(* CODESYS project Patterns of Ladderlogic programming.project

Project tree, tasks and I/O mapping:
  Device : CODESYS Control for Raspberry Pi SL, 3S - Smart Software Solutions GmbH, version 3.5.12.30
    application Application
      libraries: Standard, * (System); Util, * (System)
      task MainTask (cyclic, interval 50 ms, priority 1) calls PLC_PRG
      program PLC_PRG [LD]
      Ladder Patterns/
        Debounce/
          function block FbDebounce [LD]
        Five Rung/
          function block FbFiveRung [LD]
        Mode/
          function block FbMode [LD]
        Flasher/
          function block FbFlasher [LD]
        Mission/
          function block FbMission [LD]
        Set Reset/
          function block FbSetReset [LD]
        Reset Set/
          function block FbResetSet [LD]
        Sealed In Coil/
          function block FbSealedinCoil [LD]
        Start Stop Circuit/
          function block FbStartStopCircuit [LD]
        Input Map/
          function block FbInputMap [LD]
        State Coil Fault Coil/
          function block FbStateCoilFaultCoil [LD]
        Step/
          function block fbStep [LD]
    SoftMotion General Axis Pool
    I²C
    SPI
    GPIOs_A_B : GPIOs A/B, 3S - Smart Software Solutions GmbH, version 3.5.11.0
        unmapped channels: digital inputs (GPIO0..GPIO31), digital outputs (GPIO0..GPIO31)
    Onewire
    Camera device
      <Empty>
*)

// Device/Application/PLC_PRG
PROGRAM PLC_PRG
VAR
	SealedinCoil : FbSealedinCoil;
	xTrigger : BOOL;
	xSealedInCoil :  BOOL;
	
	
	StateCoilFaultCoil : FbStateCoilFaultCoil;
	xBreakCondition : BOOL;
	xMemoryCoil : BOOL;
	
	
	StartStopCircuit :  FbStartStopCircuit;
	xStart : BOOL;
	xStop: BOOL;
	
	
	SetReset : FbSetReset; (* use SR instead *)
	xRun : BOOL;
	xSet : BOOL;
	
	
	ResetSet : FbResetSet; (* use RS instead *)
	xReset: BOOL;
	xQs: BOOL;
	xQr: BOOL;
	
	Flasher : FbFlasher; (* use BLINK instead *)
	xFlashingLight: BOOL;
	
	
	Debounce : FbDebounce;
	xInput: BOOL;
	xInputDebounced : BOOL;
	
	
	ExtendCylinder : fbStep;
	xExtendCylinderCmd : BOOL;
	TONExtendCylinderDone : TON;
	xExtendCylinderDone: BOOL;
	tETExtend: TIME;
	RetractCylinder : fbStep;
	xRetractCylinderCmd: BOOL;
	TONRetractCylinderDone: TON;
	tETRetract: TIME;
	
	Mission : FbMission;
	xMission1Start : BOOL;
	xMission2Start : BOOL;
	xMission1Done : BOOL;
	xMission2Done : BOOL;
	xNoMission : BOOL;
	xMission1Busy : BOOL;
	xMission2Busy : BOOL;
	
	FiveRung : fbFiveRung;
	xFromSeqLogic: BOOL;
	xEStopOK: BOOL;
	xAutoMode: BOOL;
	xManMode : BOOL;
	xPushButton: BOOL;
	xSensor : BOOL;
	xResetFault: BOOL;
	xTriggerf: BOOL;
	xSafe: BOOL;
	xCommand: BOOL;
	xInPosition: BOOL;
	xTimeoutFault: BOOL;
	
	Mode : FbMode;
	xAutoModePB : BOOL;
	xManModePB : BOOL;
	xAutoSelected :BOOL;
	xManualSelected :BOOL;
	
END_VAR

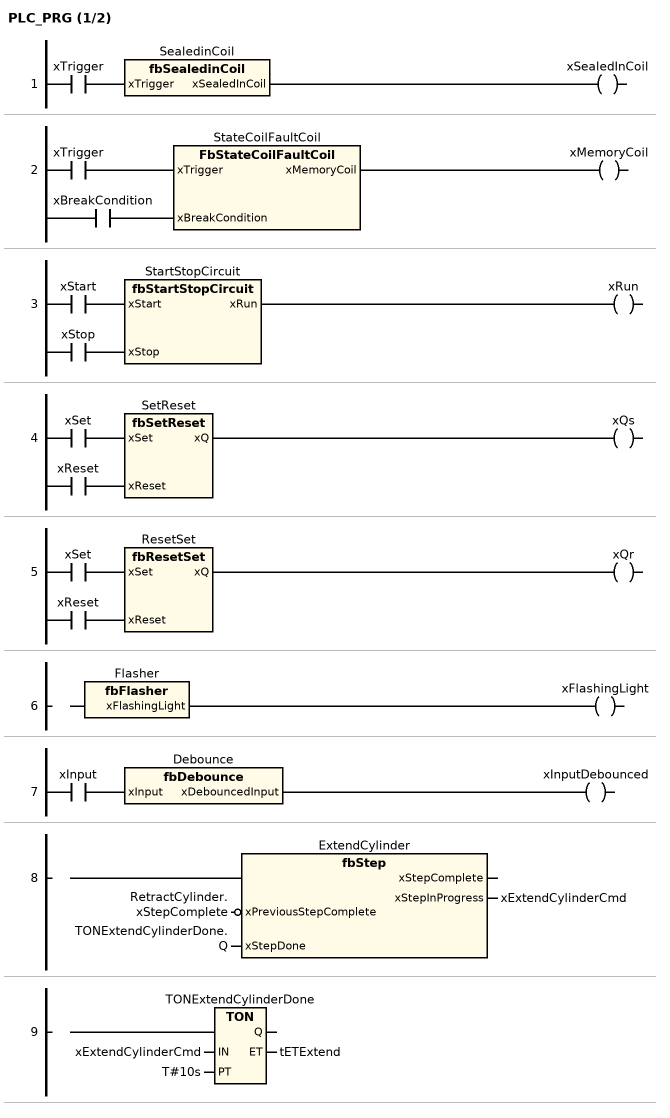
// NETWORK 1
SealedinCoil(xTrigger := xTrigger); // fbSealedinCoil
xSealedInCoil := SealedinCoil.xSealedInCoil;

// NETWORK 2
StateCoilFaultCoil(xTrigger := xTrigger, xBreakCondition := xBreakCondition); // FbStateCoilFaultCoil
xMemoryCoil := StateCoilFaultCoil.xMemoryCoil;

// NETWORK 3
StartStopCircuit(xStart := xStart, xStop := xStop); // fbStartStopCircuit
xRun := StartStopCircuit.xRun;

// NETWORK 4
SetReset(xSet := xSet, xReset := xReset); // fbSetReset
xQs := SetReset.xQ;

// NETWORK 5
ResetSet(xSet := xSet, xReset := xReset); // fbResetSet
xQr := ResetSet.xQ;

// NETWORK 6
Flasher(); // fbFlasher
xFlashingLight := Flasher.xFlashingLight;

// NETWORK 7
Debounce(xInput := xInput); // fbDebounce
xInputDebounced := Debounce.xDebouncedInput;

// NETWORK 8
ExtendCylinder(
    xPreviousStepComplete := NOT RetractCylinder.xStepComplete,
    xStepDone := TONExtendCylinderDone.Q,
    xStepInProgress => xExtendCylinderCmd); // fbStep

// NETWORK 9
TONExtendCylinderDone(IN := xExtendCylinderCmd, PT := T#10s, ET => tETExtend); // TON

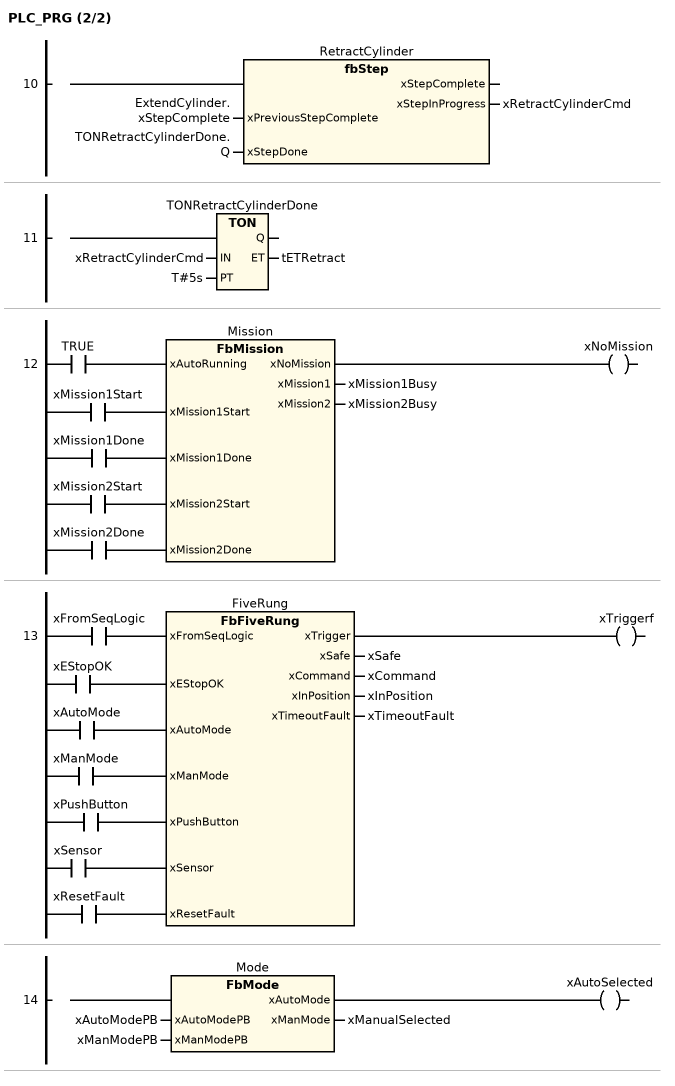
// NETWORK 10
RetractCylinder(
    xPreviousStepComplete := ExtendCylinder.xStepComplete,
    xStepDone := TONRetractCylinderDone.Q,
    xStepInProgress => xRetractCylinderCmd); // fbStep

// NETWORK 11
TONRetractCylinderDone(IN := xRetractCylinderCmd, PT := T#5s, ET => tETRetract); // TON

// NETWORK 12
Mission(
    xAutoRunning := TRUE,
    xMission1Start := xMission1Start,
    xMission1Done := xMission1Done,
    xMission2Start := xMission2Start,
    xMission2Done := xMission2Done,
    xMission1 => xMission1Busy,
    xMission2 => xMission2Busy); // FbMission
xNoMission := Mission.xNoMission;

// NETWORK 13
FiveRung(
    xFromSeqLogic := xFromSeqLogic,
    xEStopOK := xEStopOK,
    xAutoMode := xAutoMode,
    xManMode := xManMode,
    xPushButton := xPushButton,
    xSensor := xSensor,
    xResetFault := xResetFault,
    xSafe => xSafe,
    xCommand => xCommand,
    xInPosition => xInPosition,
    xTimeoutFault => xTimeoutFault); // FbFiveRung
xTriggerf := FiveRung.xTrigger;

// NETWORK 14
Mode(xAutoModePB := xAutoModePB, xManModePB := xManModePB, xManMode => xManualSelected); // FbMode
xAutoSelected := Mode.xAutoMode;

END_PROGRAM

// Device/Application/Ladder Patterns/Sealed In Coil/FbSealedinCoil
FUNCTION_BLOCK FbSealedinCoil
VAR_INPUT	
	xTrigger : BOOL;
END_VAR	
VAR_OUTPUT
	xSealedInCoil : BOOL;	
END_VAR

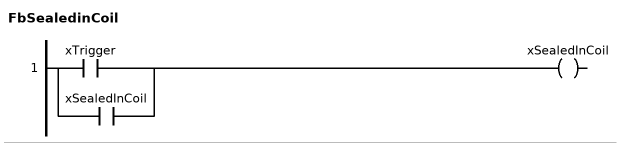
// NETWORK 1
xSealedInCoil := xTrigger OR xSealedInCoil;

END_FUNCTION_BLOCK

// Device/Application/Ladder Patterns/State Coil Fault Coil/FbStateCoilFaultCoil
FUNCTION_BLOCK FbStateCoilFaultCoil
VAR_INPUT
	xTrigger : BOOL;
	xBreakCondition: BOOL;
END_VAR
VAR_OUTPUT
	xMemoryCoil : BOOL;
END_VAR

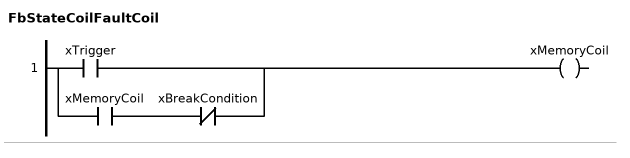
// NETWORK 1
xMemoryCoil := xTrigger OR xMemoryCoil AND NOT xBreakCondition;

END_FUNCTION_BLOCK

// Device/Application/Ladder Patterns/Start Stop Circuit/FbStartStopCircuit
FUNCTION_BLOCK FbStartStopCircuit
VAR_INPUT
	xStart : BOOL;
	xStop: BOOL;
END_VAR
VAR_OUTPUT
	xRun : BOOL;
END_VAR

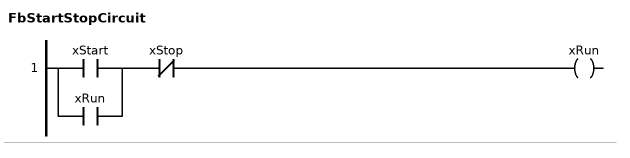
// NETWORK 1
xRun := (xStart OR xRun) AND NOT xStop;

END_FUNCTION_BLOCK

// Device/Application/Ladder Patterns/Set Reset/FbSetReset
FUNCTION_BLOCK FbSetReset (* set dominant Flip Flop *)
(* Use of this pattern is *NOT* recommended => suggest use of SR (FB) from Standard lib instead *)
VAR_INPUT
	xSet : BOOL;
	xReset : BOOL;
END_VAR
VAR_OUTPUT
	xQ : BOOL;(* Memory *)
END_VAR

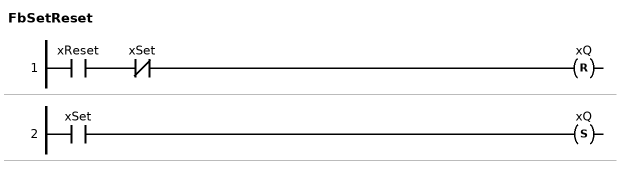
// NETWORK 1
xQ R= xReset AND NOT xSet;

// NETWORK 2
xQ S= xSet;

END_FUNCTION_BLOCK

// Device/Application/Ladder Patterns/Reset Set/FbResetSet
FUNCTION_BLOCK FbResetSet (* Reset dominant Flip Flop*)
(* Use of this pattern is *NOT* recommended => suggest use of RS (FB) from Standard lib instead *)
VAR_INPUT
	xSet : BOOL;
	xReset : BOOL;
END_VAR
VAR_OUTPUT
	xQ : BOOL;(* Memory *)
END_VAR

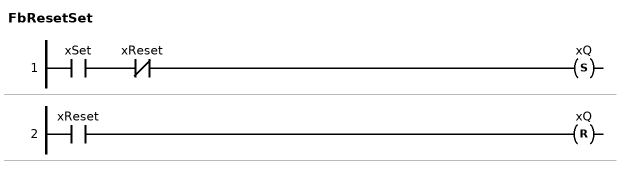
// NETWORK 1
xQ S= xSet AND NOT xReset;

// NETWORK 2
xQ R= xReset;

END_FUNCTION_BLOCK

// Device/Application/Ladder Patterns/Flasher/FbFlasher
(* Use of this pattern is *NOT* recommended *)
FUNCTION_BLOCK FbFlasher  
VAR
	(* pattern original *)
	Timer1 : Ton;
	tET1 : TIME;
	Timer2 : Ton;
	tET2: TIME;
	
	(* IEC standard alternative *)
	BLINK : util.BLINK;
	xBlink: BOOL;
END_VAR
VAR_OUTPUT
	xFlashingLight : BOOL;
END_VAR

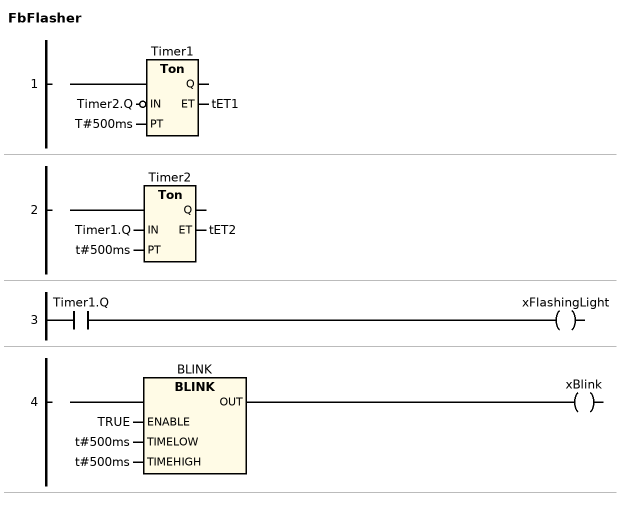
// NETWORK 1
Timer1(IN := NOT Timer2.Q, PT := T#500ms, ET => tET1); // Ton

// NETWORK 2
Timer2(IN := Timer1.Q, PT := t#500ms, ET => tET2); // Ton

// NETWORK 3
xFlashingLight := Timer1.Q;

// NETWORK 4
BLINK(ENABLE := TRUE, TIMELOW := t#500ms, TIMEHIGH := t#500ms);
xBlink := BLINK.OUT;

END_FUNCTION_BLOCK

// Device/Application/Ladder Patterns/Debounce/FbDebounce
(* Due to an increase in the use of solid-state sensors like proximity switches, this pattern will be less likely to be seen *)
FUNCTION_BLOCK FbDebounce  
VAR_INPUT
	xInput : BOOL;
END_VAR
VAR_OUTPUT
	xDebouncedInput : BOOL;
END_VAR
VAR
	DelayOn : Ton;
	tETon : TIME;
	DelayOff : Ton;
	tEToff: TIME;
END_VAR

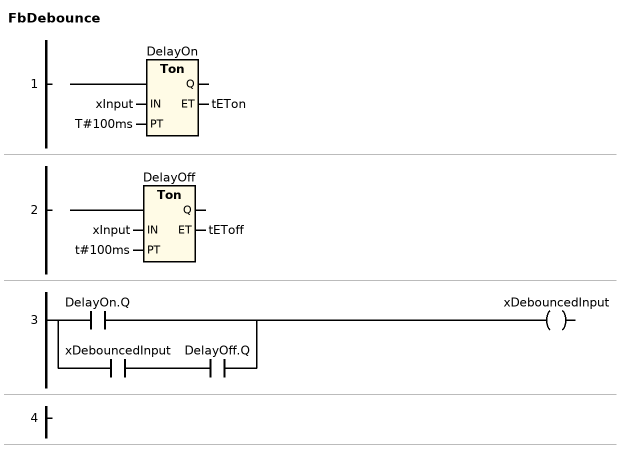
// NETWORK 1
DelayOn(IN := xInput, PT := T#100ms, ET => tETon); // Ton

// NETWORK 2
DelayOff(IN := xInput, PT := t#100ms, ET => tEToff); // Ton

// NETWORK 3
xDebouncedInput := DelayOn.Q OR xDebouncedInput AND DelayOff.Q;

// NETWORK 4

END_FUNCTION_BLOCK

// Device/Application/Ladder Patterns/Step/fbStep
FUNCTION_BLOCK fbStep
VAR_INPUT
	xPreviousStepComplete : BOOL; (* // previous step completed *)
	xStepDone : BOOL; (* Step should stay active until this flag is set TRUE *)
END_VAR
VAR_OUTPUT
	xStepComplete : BOOL; (* Until external logic signals "done", this step status is FALSE, if the external logic signals done, this step is completed *)
	xStepInProgress : BOOL; (* This flag should be used to steer a codition *)
END_VAR

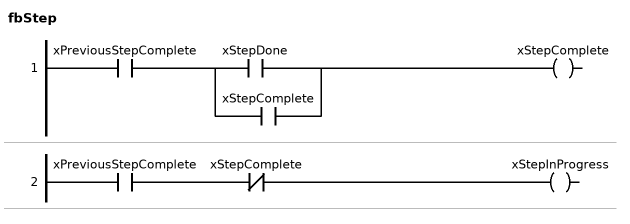
// NETWORK 1
xStepComplete := xPreviousStepComplete AND (xStepDone OR xStepComplete);

// NETWORK 2
xStepInProgress := xPreviousStepComplete AND NOT xStepComplete;

END_FUNCTION_BLOCK

// Device/Application/Ladder Patterns/Mission/FbMission
FUNCTION_BLOCK FbMission
VAR_INPUT
	xAutoRunning : BOOL;
	xMission1Start : BOOL;
	xMission1Done : BOOL;
	xMission2Start : BOOL;
	xMission2Done : BOOL;
END_VAR
VAR_OUTPUT	
	xNoMission : BOOL;
	xMission1 : BOOL; (* Busy 1 *)
	xMission2 : BOOL; (* Busy 2 *)
END_VAR

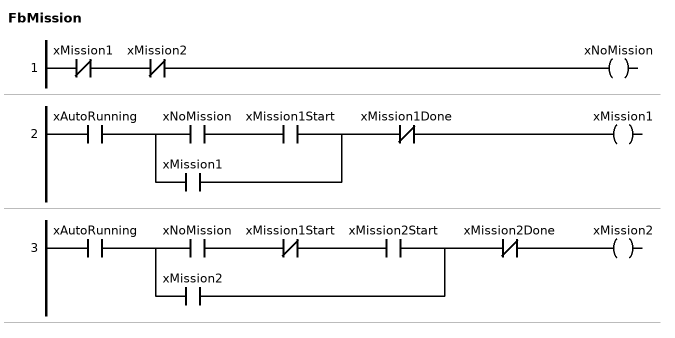
// NETWORK 1
xNoMission := NOT xMission1 AND NOT xMission2;

// NETWORK 2
xMission1 := xAutoRunning AND (xNoMission AND xMission1Start OR xMission1) AND NOT xMission1Done;

// NETWORK 3
xMission2 := xAutoRunning AND (xNoMission AND NOT xMission1Start AND xMission2Start OR xMission2) AND NOT xMission2Done;

END_FUNCTION_BLOCK

// Device/Application/Ladder Patterns/Five Rung/FbFiveRung
FUNCTION_BLOCK FbFiveRung
VAR_INPUT
	xFromSeqLogic: BOOL;
	xEStopOK: BOOL;
	xAutoMode: BOOL;
	xManMode : BOOL;
	xPushButton: BOOL;
	xSensor : BOOL;
	xResetFault: BOOL;
END_VAR
VAR_OUTPUT
	xTrigger: BOOL;
	xSafe: BOOL;
	xCommand: BOOL;
	xInPosition: BOOL;
	xTimeoutFault: BOOL;
END_VAR
VAR
	FaultTimer: TON;
	tETFault: TIME;	
END_VAR

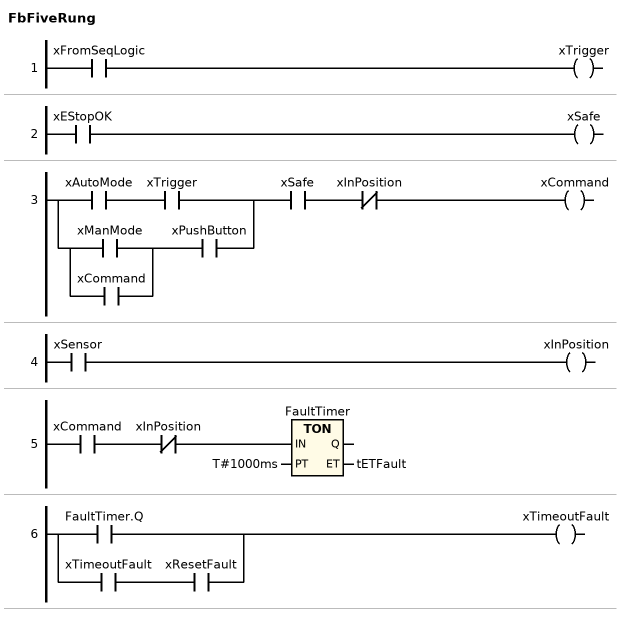
// NETWORK 1
xTrigger := xFromSeqLogic;

// NETWORK 2
xSafe := xEStopOK;

// NETWORK 3
xCommand := (xAutoMode AND xTrigger OR (xManMode OR xCommand) AND xPushButton) AND xSafe AND NOT xInPosition;

// NETWORK 4
xInPosition := xSensor;

// NETWORK 5
FaultTimer(IN := xCommand AND NOT xInPosition, PT := T#1000ms, ET => tETFault); // TON

// NETWORK 6
xTimeoutFault := FaultTimer.Q OR xTimeoutFault AND xResetFault;

END_FUNCTION_BLOCK

// Device/Application/Ladder Patterns/Mode/FbMode
FUNCTION_BLOCK FbMode
VAR_INPUT
	xAutoModePB : BOOL;
	xManModePB : BOOL;
END_VAR
VAR_OUTPUT
	xAutoMode : BOOL;
	xManMode : BOOL;
END_VAR

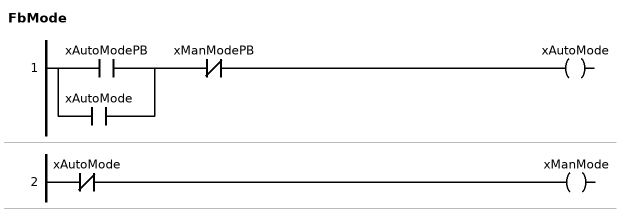
// NETWORK 1
xAutoMode := (xAutoModePB OR xAutoMode) AND NOT xManModePB;

// NETWORK 2
xManMode := NOT xAutoMode;

END_FUNCTION_BLOCK

// Device/Application/Ladder Patterns/Input Map/FbInputMap
FUNCTION_BLOCK FbInputMap (* IO mapping *)
(*
	Use of this pattern is PLC-specific, for CODESYS3 (thus TwinCAT3) it is obselete.
 
	For instance, Beckhoff’s TwinCAT PLC software already includes an I/O mapping function, 
	so you map internal variables like MyMachine.MotorRunning to a physical input using their System Manager. 
	Their I/O scan is also synchronous to the program scan, so there are fewer advantages to using the Input Map pattern with Beckhoff TwinCAT systems.
*)
VAR
	xInput : BOOL;
	xA : BOOL;
	xB : BOOL;
END_VAR

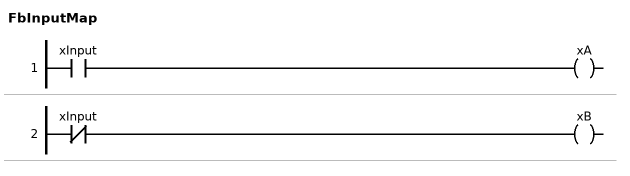
// NETWORK 1
xA := xInput;

// NETWORK 2
xB := NOT xInput;

END_FUNCTION_BLOCK
